(* PLC project CoDeSys External Library Template, WAGO e!COCKPIT e!COCKPIT, author 3S - Smart Software Solutions GmbH *)
(* stored: creationDateTime 2019-10-29T12:37:19.4496817, version 3.5.5.30, modificationDateTime 2019-10-29T12:36:39.3744516, organization 3S - Smart Software Solutions GmbH *)
(* Library project template with all possible element types, docu and a sample project structure *)

{attribute 'qualified_only'}
{attribute 'strict'}
TYPE enumPPPSUrzadenieStatus : (Nieaktywny := 1, Oczekiwanie := 2, Prawidlowy := 3, Ostrzezenie := 4, Awaria := 5, Krytyczny := 6);
END_TYPE
